(*
SPDX-FileCopyrightText: © 2026 Oleksandr Tiutyk <trofimich@gmail.com>
SPDX-License-Identifier: MIT
License: https://opensource.org/license/mit
*)

{attribute 'no_explicit_call' := 'Direct call is not allowed'} 
FUNCTION_BLOCK AutomaticJsonSerializer EXTENDS TOF_Core.Object
VAR
	{attribute 'hide'} 
	_ClassName : STRING := __POUNAME();
	
	_JsonSaxWriter : Tc3_JsonXml.FB_JsonSaxWriter;
	_JsonDataTypeWriter : Tc3_JsonXml.FB_JsonReadWriteDatatype;
END_VAR

{attribute 'monitoring' := 'call'}
PROPERTY ClassName : REFERENCE TO STRING
GET
ClassName REF= _ClassName;
END_GET
END_PROPERTY

METHOD CreateJsonFromStructure
VAR_INPUT
	sourceStructure : ANY;
	extender : IJsonExtender := 0;
END_VAR
VAR_IN_OUT CONSTANT
    targetJson : TOF_Core.JSON_DOCUMENT;
END_VAR
VAR_OUTPUT
	jsonSize : UDINT; 
END_VAR
InternalCreateJsonFromStructure(sourceStructure, extender, targetJson, jsonSize => jsonSize);
END_METHOD

METHOD CreateJsonFromStructureByVarInfo
VAR_INPUT
	sourceStructureVarInfo : __SYSTEM.VAR_INFO;
	extender : IJsonExtender := 0;
END_VAR
VAR_IN_OUT CONSTANT
    targetJson : TOF_Core.JSON_DOCUMENT;
END_VAR
VAR_OUTPUT
	jsonSize : UDINT; 
END_VAR
VAR
	argumentNullException : TOF_Core.ArgumentNotSpecifiedException;
	argumentTypeNotSupportedException : TOF_Core.ArgumentTypeNotSupportedException;
	standardException : TOF_Core.StandardException;
	
	errorCode : HRESULT;
END_VAR
IF sourceStructureVarInfo.ByteAddress = 0 THEN
	argumentNullException.Throw(NamespaceName, ClassName, __POUNAME(), __POSITION(), 'sourceStructureVarInfo');
END_IF

IF sourceStructureVarInfo.TypeClass <> __SYSTEM.TYPE_CLASS.TYPE_USERDEF THEN
	argumentTypeNotSupportedException.Throw(NamespaceName, ClassName, __POUNAME(), __POSITION(), 'sourceStructureVarInfo', sourceStructureVarInfo.TypeClass);
END_IF

_JsonSaxWriter.ResetDocument();

IF extender <> 0 THEN
	extender.ExtendAtStart(_JsonSaxWriter);
END_IF

IF NOT _JsonDataTypeWriter.AddJsonValueFromSymbol(_JsonSaxWriter, sourceStructureVarInfo.TypeName, TO_UDINT(sourceStructureVarInfo.BitSize / 8), sourceStructureVarInfo.ByteAddress, hrErrorCode => errorCode) THEN
	standardException.Throw(NamespaceName, ClassName, __POUNAME(), __POSITION(), TOF_Core.WideStrings.Concat255("Can't generate JSON representation from the symbol of type '", TO_WSTRING(sourceStructureVarInfo.TypeName), "'"), TO_UDINT(errorCode));
END_IF

IF extender <> 0 THEN
	extender.ExtendAtFinish(_JsonSaxWriter);
END_IF

jsonSize := _JsonSaxWriter.CopyDocument(targetJson, SIZEOF(targetJson), hrErrorCode => errorCode);

IF errorCode <> 0 THEN
	standardException.Throw(NamespaceName, ClassName, __POUNAME(), __POSITION(), TOF_Core.WideStrings.Concat255("Can't fill JSON from the symbol of type '", TO_WSTRING(sourceStructureVarInfo.TypeName), "'"), TO_UDINT(errorCode));
END_IF
END_METHOD

{attribute 'monitoring' := 'call'}
PROPERTY DecimalPlaces : DINT
GET
DecimalPlaces := _JsonSaxWriter.GetMaxDecimalPlaces();
END_GET
SET
_JsonSaxWriter.SetMaxDecimalPlaces(DecimalPlaces);
END_SET
END_PROPERTY

METHOD FillStructureByVarInfoFromJson
VAR_IN_OUT CONSTANT
	json : TOF_Core.JSON_DOCUMENT;	
END_VAR
VAR_INPUT
	targetStructureVarInfo : __SYSTEM.VAR_INFO;
END_VAR
VAR
	argumentNullException : TOF_Core.ArgumentNotSpecifiedException;
	argumentTypeNotSupportedException : TOF_Core.ArgumentTypeNotSupportedException;
	standardException : TOF_Core.StandardException;
	
	structureTypeName : STRING;	 
	errorCode : HRESULT;
END_VAR
IF targetStructureVarInfo.ByteAddress = 0 THEN
	argumentNullException.Throw(NamespaceName, ClassName, __POUNAME(), __POSITION(), 'targetStructureVarInfo');
END_IF

IF targetStructureVarInfo.TypeClass <> __SYSTEM.TYPE_CLASS.TYPE_USERDEF THEN
	argumentTypeNotSupportedException.Throw(NamespaceName, ClassName, __POUNAME(), __POSITION(), 'targetStructureVarInfo', targetStructureVarInfo.TypeClass);
END_IF

structureTypeName := _JsonDataTypeWriter.GetDatatypeNameByAddress(TO_UDINT(targetStructureVarInfo.BitSize / 8), targetStructureVarInfo.ByteAddress, hrErrorCode => errorCode);

IF errorCode <> 0 THEN
	standardException.Throw(NamespaceName, ClassName, __POUNAME(), __POSITION(), "Can't get structure type of the target structure", TO_UDINT(errorCode));
END_IF

_JsonDataTypeWriter.SetSymbolFromJson(json, structureTypeName, TO_UDINT(targetStructureVarInfo.BitSize / 8), targetStructureVarInfo.ByteAddress, hrErrorCode => errorCode);

IF errorCode <> 0 THEN
	standardException.Throw(NamespaceName, ClassName, __POUNAME(), __POSITION(), "Can't fill target structure by specified json document", TO_UDINT(errorCode));
END_IF
END_METHOD

METHOD FillStructureFromJson
VAR_IN_OUT CONSTANT
	json : TOF_Core.JSON_DOCUMENT;	
END_VAR
VAR_INPUT
	targetStructure : ANY;
END_VAR
InternalFillStructureFromJson(json, targetStructure);
END_METHOD

METHOD PROTECTED InternalCreateJsonFromStructure
VAR_INPUT
	sourceStructure : __SYSTEM.AnyType;
	extender : IJsonExtender := 0;
END_VAR
VAR_IN_OUT CONSTANT
    targetJson : TOF_Core.JSON_DOCUMENT;
END_VAR
VAR_OUTPUT
	jsonSize : UDINT; 
END_VAR
VAR
	argumentNullException : TOF_Core.ArgumentNotSpecifiedException;
	argumentTypeNotSupportedException : TOF_Core.ArgumentTypeNotSupportedException;
	standardException : TOF_Core.StandardException;
	
	structureTypeName : STRING;	 
	errorCode : HRESULT;
END_VAR
IF sourceStructure.pValue = 0 THEN
	argumentNullException.Throw(NamespaceName, ClassName, __POUNAME(), __POSITION(), 'sourceStructure');
END_IF

IF sourceStructure.TypeClass <> __SYSTEM.TYPE_CLASS.TYPE_USERDEF THEN
	argumentTypeNotSupportedException.Throw(NamespaceName, ClassName, __POUNAME(), __POSITION(), 'sourceStructure', sourceStructure.TypeClass);
END_IF

_JsonSaxWriter.ResetDocument();

structureTypeName := _JsonDataTypeWriter.GetDatatypeNameByAddress(TO_UDINT(sourceStructure.diSize), sourceStructure.pValue, hrErrorCode => errorCode);

IF errorCode <> 0 THEN
	standardException.Throw(NamespaceName, ClassName, __POUNAME(), __POSITION(), "Can't get structure type of the source structure", TO_UDINT(errorCode));
END_IF

IF extender <> 0 THEN
	extender.ExtendAtStart(_JsonSaxWriter);
END_IF

IF NOT _JsonDataTypeWriter.AddJsonValueFromSymbol(_JsonSaxWriter, structureTypeName, TO_UDINT(sourceStructure.diSize), sourceStructure.pValue, hrErrorCode => errorCode) THEN
	standardException.Throw(NamespaceName, ClassName, __POUNAME(), __POSITION(), TOF_Core.WideStrings.Concat255("Can't generate JSON representation from the symbol of type '", TO_WSTRING(structureTypeName), "'"), TO_UDINT(errorCode));
END_IF

IF extender <> 0 THEN
	extender.ExtendAtFinish(_JsonSaxWriter);
END_IF

jsonSize := _JsonSaxWriter.CopyDocument(targetJson, SIZEOF(targetJson), hrErrorCode => errorCode);

IF errorCode <> 0 THEN
	standardException.Throw(NamespaceName, ClassName, __POUNAME(), __POSITION(), TOF_Core.WideStrings.Concat255("Can't fill JSON from the symbol of type '", TO_WSTRING(structureTypeName), "'"), TO_UDINT(errorCode));
END_IF
END_METHOD

METHOD PROTECTED InternalFillStructureFromJson
VAR_IN_OUT CONSTANT
	json : TOF_Core.JSON_DOCUMENT;	
END_VAR
VAR_INPUT
	targetStructure : __SYSTEM.AnyType;
END_VAR
VAR
	argumentNullException : TOF_Core.ArgumentNotSpecifiedException;
	argumentTypeNotSupportedException : TOF_Core.ArgumentTypeNotSupportedException;
	standardException : TOF_Core.StandardException;
	
	structureTypeName : STRING;	 
	errorCode : HRESULT;
END_VAR
IF targetStructure.pValue = 0 THEN
	argumentNullException.Throw(NamespaceName, ClassName, __POUNAME(), __POSITION(), 'targetStructure');
END_IF

IF targetStructure.TypeClass <> __SYSTEM.TYPE_CLASS.TYPE_USERDEF THEN
	argumentTypeNotSupportedException.Throw(NamespaceName, ClassName, __POUNAME(), __POSITION(), 'targetStructure', targetStructure.TypeClass);
END_IF

structureTypeName := _JsonDataTypeWriter.GetDatatypeNameByAddress(TO_UDINT(targetStructure.diSize), targetStructure.pValue, hrErrorCode => errorCode);

IF errorCode <> 0 THEN
	standardException.Throw(NamespaceName, ClassName, __POUNAME(), __POSITION(), "Can't get structure type of the target structure", TO_UDINT(errorCode));
END_IF

_JsonDataTypeWriter.SetSymbolFromJson(json, structureTypeName, TO_UDINT(targetStructure.diSize), targetStructure.pValue, hrErrorCode => errorCode);

IF errorCode <> 0 THEN
	standardException.Throw(NamespaceName, ClassName, __POUNAME(), __POSITION(), "Can't fill target structure by specified json document", TO_UDINT(errorCode));
END_IF
END_METHOD

{attribute 'monitoring' := 'call'}
PROPERTY NamespaceName : REFERENCE TO STRING
GET
NamespaceName REF= CurrentNamespace.Name;
END_GET
END_PROPERTY

{attribute 'monitoring' := 'call'}
PROPERTY SelfSize : ULINT
GET
SelfSize := XSIZEOF(THIS^);
END_GET
END_PROPERTY

METHOD PRIVATE SetFormatOptions
VAR_INPUT
	decimalPlaces : BYTE := 10;
	formatOptions : EJsonPrettyFormatOptions := EJsonPrettyFormatOptions.eFormatSingleLineArray;
	identChar : SINT := 9;
	identCharCount : BYTE := 1;
END_VAR
_JsonSaxWriter.SetMaxDecimalPlaces(decimalPlaces);
END_METHOD

{attribute 'TcRpcEnable':='1'}
METHOD TryCreateJsonFromStructure : BOOL
VAR_INPUT
	sourceStructure : ANY;
	extender : IJsonExtender := 0;
END_VAR
VAR_IN_OUT CONSTANT
    targetJson : TOF_Core.JSON_DOCUMENT;
END_VAR
VAR_OUTPUT
	jsonSize : UDINT; 
END_VAR
__TRY
	InternalCreateJsonFromStructure(sourceStructure, extender, targetJson, jsonSize => jsonSize);

	TryCreateJsonFromStructure := TRUE;
__CATCH
__ENDTRY
END_METHOD

METHOD TryCreateJsonFromStructureByVarInfo : BOOL
VAR_INPUT
	sourceStructureVarInfo : __SYSTEM.VAR_INFO;
	extender : IJsonExtender := 0;
END_VAR
VAR_IN_OUT CONSTANT
    targetJson : TOF_Core.JSON_DOCUMENT;
END_VAR
VAR_OUTPUT
	jsonSize : UDINT; 
END_VAR
__TRY
	CreateJsonFromStructureByVarInfo(sourceStructureVarInfo, extender, targetJson, jsonSize => jsonSize);
	
	TryCreateJsonFromStructureByVarInfo := TRUE;
__CATCH
__ENDTRY
END_METHOD

METHOD TryFillStructureByVarInfoFromJson : BOOL
VAR_IN_OUT CONSTANT
	json : TOF_Core.JSON_DOCUMENT;	
END_VAR
VAR_INPUT
	targetStructureVarInfo : __SYSTEM.VAR_INFO;
END_VAR
__TRY
	FillStructureByVarInfoFromJson(json, targetStructureVarInfo);
	
	TryFillStructureByVarInfoFromJson := TRUE;
__CATCH	
__ENDTRY
END_METHOD

METHOD TryFillStructureFromJson : BOOL
VAR_IN_OUT CONSTANT
	json : TOF_Core.JSON_DOCUMENT;	
END_VAR
VAR_INPUT
	targetStructure : ANY;
END_VAR
__TRY
	InternalFillStructureFromJson(json, targetStructure);
	
	TryFillStructureFromJson := TRUE;
__CATCH
__ENDTRY
END_METHOD

END_FUNCTION_BLOCK

(* stored: Version 1.1.0.1
   POU AutomaticJsonSerializer: Id {a4623321-e5e2-4514-b5b7-6f50c93efdb9}, SpecialFunc None
   Folder Service memebers: Id {ac3ba484-d0b1-4d7e-b557-cd243c8b8997}
   Property ClassName: Id {0ef034e0-c59c-400d-8910-5199a1e43c28}
   Get Get: Id {7d8e441f-d9e1-4fe6-a84f-2d3a88ae1b83}
   Method CreateJsonFromStructure: Id {defd30bb-3636-4b3d-a29d-4ee5f3966212}
   Method CreateJsonFromStructureByVarInfo: Id {d6f652b9-17a4-4ec4-936c-676a73e01a2d}
   Property DecimalPlaces: Id {856a998f-c63b-4bfb-be2d-ebc0ce7cf745}
   Get Get: Id {94eff383-c1b9-45b7-8cbb-da0c6c3a2aac}
   Set Set: Id {e5e3c1bb-4425-43f2-a416-2b4fee3a3ddc}
   Method FillStructureByVarInfoFromJson: Id {3b0559f7-3cc9-4407-b03c-9992acf72583}
   Method FillStructureFromJson: Id {b53042c3-1eea-4151-a973-f56939241dea}
   Method InternalCreateJsonFromStructure: Id {828ddc06-4e4b-4f22-bd8f-3234f73fd728}
   Method InternalFillStructureFromJson: Id {cd668581-fbff-4bb3-b0d3-914c47132fdf}
   Property NamespaceName: Id {7371ecef-1936-4268-af0d-813ed5877183}
   Get Get: Id {a712aceb-e580-4469-b321-74f0e6ab0c97}
   Property SelfSize: Id {4e2cc4a2-86a6-48cc-a757-58f1b82e3903}
   Get Get: Id {3c9a353a-dae3-4a6a-8486-44c6e5bd0b57}
   Method SetFormatOptions: Id {c6cdde79-cf05-4b34-97ff-f0f4810b70ea}
   Method TryCreateJsonFromStructure: Id {35373f3b-1087-4a79-950c-0b141211bf99}
   Method TryCreateJsonFromStructureByVarInfo: Id {486e285a-fcfe-44f3-9023-743f121d8975}
   Method TryFillStructureByVarInfoFromJson: Id {25972cd3-eceb-4afa-aeb2-ef7585c39b37}
   Method TryFillStructureFromJson: Id {b5b62249-7ff4-4c95-ba2a-e43e9757d053} *)
